(* PLC project MotionTest1, Higen MCL 1 *)
(* stored: creationDateTime 2012-01-06T15:20:13, modificationDateTime 2026-03-16T00:20:08 *)

PROGRAM main
  VAR
    clock : ULINT;
    Done : BOOL;
    PosAxis : AXIS_REF;
    NegAxis : AXIS_REF;
    moveA : MC_MoveAbsolute;
    switch : MC_Power;
    readpos : MC_ReadActualPosition;
    PnNeg : LREAL;
    PnPos : LREAL;
    JPOpos : LREAL;
    JPOneg : LREAL;
    AccPos : LREAL;
    AccNeg : LREAL;
    VnNeg : LREAL;
    VnPos : LREAL;
    setpos : MC_SetPosition;
    readspeed : MC_ReadParameter;
    my_simulated_axis : MC_Sim;
    MC_MoveContinuousAbsolute0 : MC_MoveContinuousAbsolute;
    MC_MoveAbsolute0 : MC_MoveAbsolute;
    MC_Power0 : MC_Power;
    MC_ReadActualPosition0 : MC_ReadActualPosition;
    MC_SetPosition0 : MC_SetPosition;
    MC_ReadParameter0 : MC_ReadParameter;
    MC_Sim0 : MC_Sim;
    MC_MoveContinuousAbsolute1 : MC_MoveContinuousAbsolute;
    MC_MoveContinuousAbsolute2 : MC_MoveContinuousAbsolute;
    MC_MoveContinuousAbsolute3 : MC_MoveContinuousAbsolute;
    MC_ReadParameter1 : MC_ReadParameter;
    MC_ReadParameter2 : MC_ReadParameter;
    MC_ReadParameter3 : MC_ReadParameter;
    MC_ReadParameter4 : MC_ReadParameter;
    MC_SetOverride0 : MC_SetOverride;
    MC_SetOverride1 : MC_SetOverride;
  END_VAR

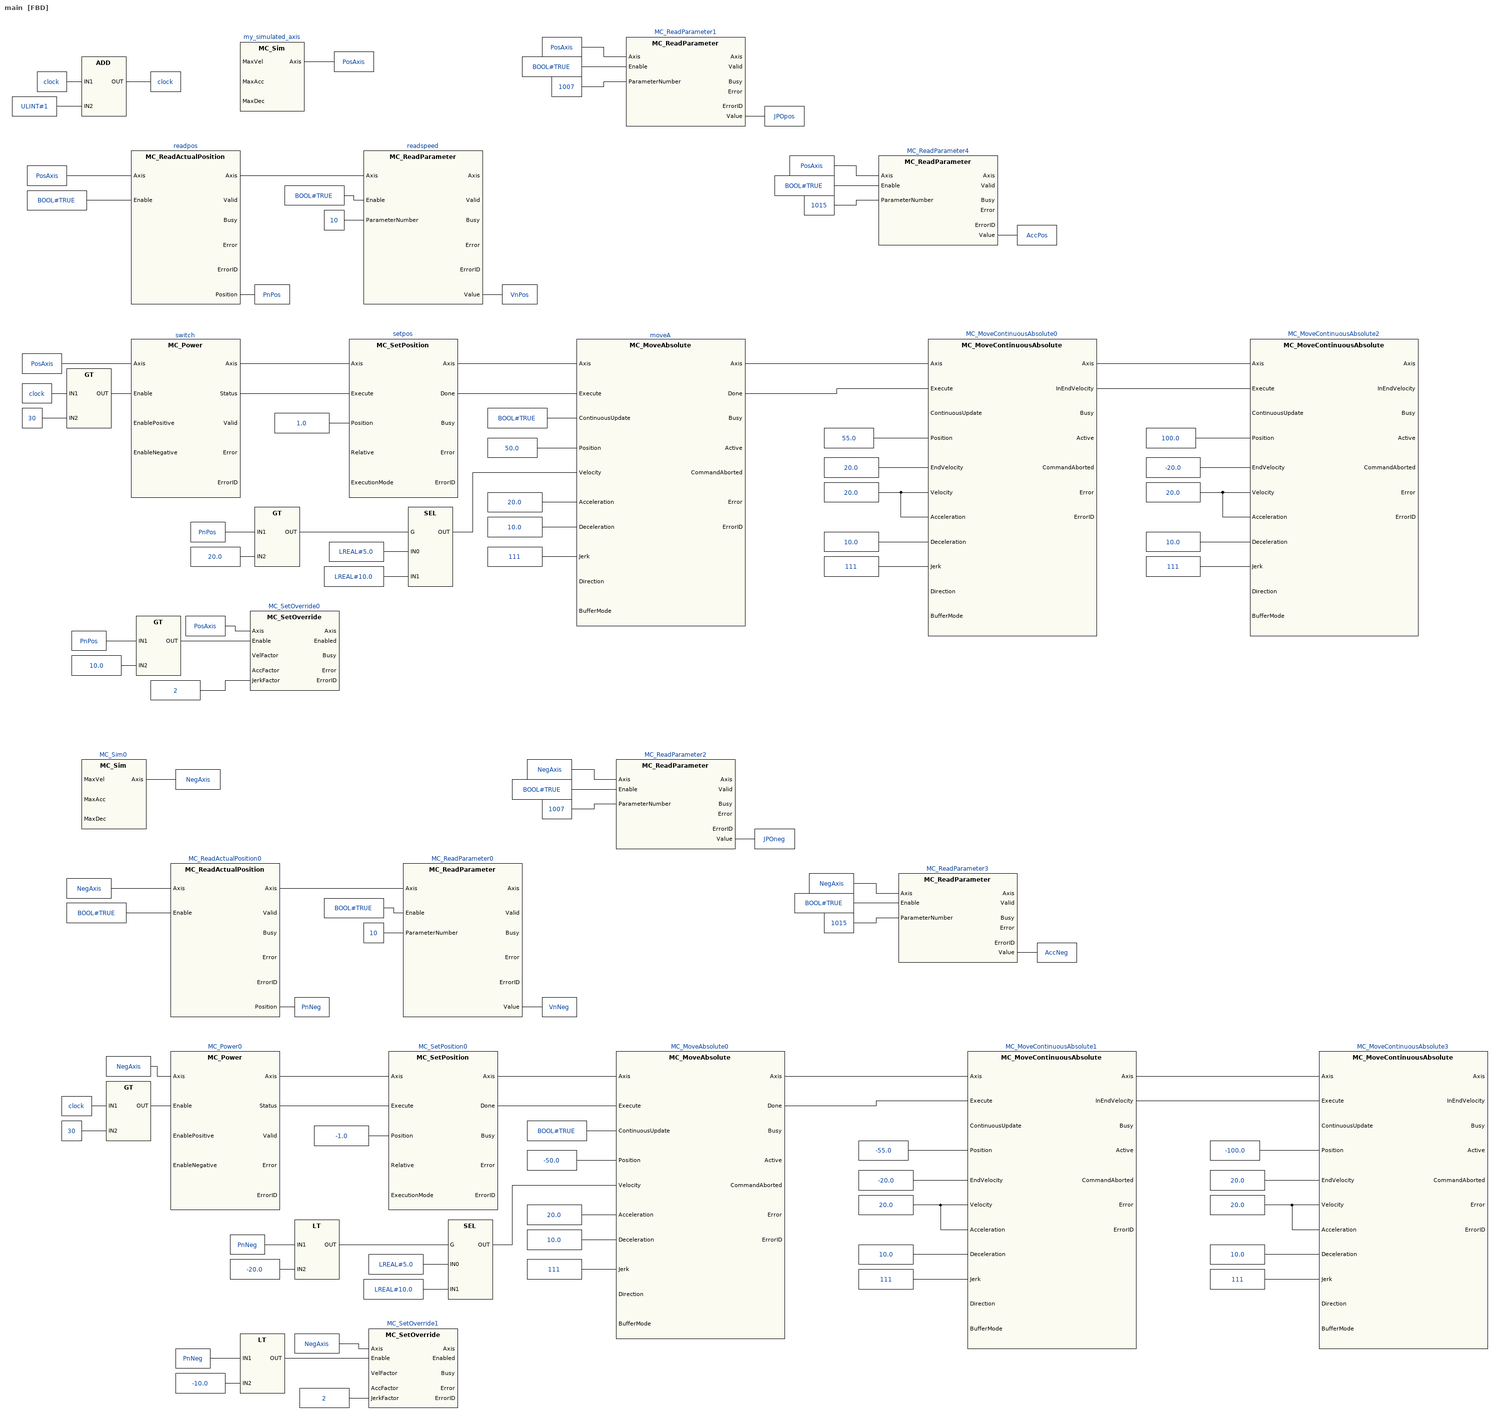
(* FBD diagram, written out as Structured Text *)
clock := clock + ULINT#1;
readpos(Axis := PosAxis, Enable := BOOL#TRUE);
PnPos := readpos.Position;
readspeed(Axis := readpos.Axis, Enable := BOOL#TRUE, ParameterNumber := 10);
VnPos := readspeed.Value;
my_simulated_axis();
PosAxis := my_simulated_axis.Axis;
MC_ReadActualPosition0(Axis := NegAxis, Enable := BOOL#TRUE);
PnNeg := MC_ReadActualPosition0.Position;
MC_ReadParameter0(Axis := MC_ReadActualPosition0.Axis, Enable := BOOL#TRUE, ParameterNumber := 10);
VnNeg := MC_ReadParameter0.Value;
MC_Sim0();
NegAxis := MC_Sim0.Axis;
MC_ReadParameter1(Axis := PosAxis, Enable := BOOL#TRUE, ParameterNumber := 1007);
JPOpos := MC_ReadParameter1.Value;
MC_ReadParameter2(Axis := NegAxis, Enable := BOOL#TRUE, ParameterNumber := 1007);
JPOneg := MC_ReadParameter2.Value;
MC_ReadParameter3(Axis := NegAxis, Enable := BOOL#TRUE, ParameterNumber := 1015);
AccNeg := MC_ReadParameter3.Value;
MC_ReadParameter4(Axis := PosAxis, Enable := BOOL#TRUE, ParameterNumber := 1015);
AccPos := MC_ReadParameter4.Value;
switch(Axis := PosAxis, Enable := clock > 30);
setpos(Axis := switch.Axis, Execute := switch.Status, Position := 1.0);
moveA(Axis := setpos.Axis, Execute := setpos.Done, ContinuousUpdate := BOOL#TRUE, Position := 50.0, Velocity := SEL(PnPos > 20.0, LREAL#5.0, LREAL#10.0), Acceleration := 20.0, Deceleration := 10.0, Jerk := 111);
MC_MoveContinuousAbsolute0(Axis := moveA.Axis, Execute := moveA.Done, Position := 55.0, EndVelocity := 20.0, Velocity := 20.0, Acceleration := 20.0, Deceleration := 10.0, Jerk := 111);
MC_Power0(Axis := NegAxis, Enable := clock > 30);
MC_SetPosition0(Axis := MC_Power0.Axis, Execute := MC_Power0.Status, Position := -1.0);
MC_MoveAbsolute0(Axis := MC_SetPosition0.Axis, Execute := MC_SetPosition0.Done, ContinuousUpdate := BOOL#TRUE, Position := -50.0, Velocity := SEL(PnNeg < (-20.0), LREAL#5.0, LREAL#10.0), Acceleration := 20.0, Deceleration := 10.0, Jerk := 111);
MC_MoveContinuousAbsolute1(Axis := MC_MoveAbsolute0.Axis, Execute := MC_MoveAbsolute0.Done, Position := -55.0, EndVelocity := -20.0, Velocity := 20.0, Acceleration := 20.0, Deceleration := 10.0, Jerk := 111);
MC_MoveContinuousAbsolute2(Axis := MC_MoveContinuousAbsolute0.Axis, Execute := MC_MoveContinuousAbsolute0.InEndVelocity, Position := 100.0, EndVelocity := -20.0, Velocity := 20.0, Acceleration := 20.0, Deceleration := 10.0, Jerk := 111);
MC_MoveContinuousAbsolute3(Axis := MC_MoveContinuousAbsolute1.Axis, Execute := MC_MoveContinuousAbsolute1.InEndVelocity, Position := -100.0, EndVelocity := 20.0, Velocity := 20.0, Acceleration := 20.0, Deceleration := 10.0, Jerk := 111);
MC_SetOverride0(Axis := PosAxis, Enable := PnPos > 10.0, JerkFactor := 2);
MC_SetOverride1(Axis := NegAxis, Enable := PnNeg < (-10.0), JerkFactor := 2);
END_PROGRAM

CONFIGURATION conf
  RESOURCE res ON PLC
    TASK milisecond(INTERVAL := T#10ms, PRIORITY := 0);
    PROGRAM maininstance WITH milisecond : main;
  END_RESOURCE
END_CONFIGURATION
